(* Logix 5000 project; controller Motor_Test vendor 1 type 14 code 155 rev 32.11; software revision 32.01 *)

TASK MainTask (continuous, watchdog 500 ms) : MainProgram

MODULES
   Local : vendor 1 type 14 code 155 (PointIO 0, rev 32.11)
      Discrete_IO : Embedded (PointIO 1, rev 32.11, Output RPI 20 ms)
END_MODULES

VAR_GLOBAL   (* controller tags *)
   Empty : BOOL;
   Full : BOOL;
   Level : COUNTER := (PRE := 3, ACC := 1);
   LoadBegin : BOOL;
   LoadDone : BOOL;
   MoveSlots : DINT;
   OPC : BOOL;
   Slot : COUNTER := (PRE := 20, ACC := 1);
   TotalSteps : COUNTER := (PRE := 200);
END_VAR

PROGRAM MainProgram   (* main routine MainRoutine *)
VAR
   Begin_Step : BOOL;
   Change : BOOL;
   Count : COUNTER := (PRE := 10);
   DIR_Change : BOOL;
   Direction_CCW : ALIAS FOR Local:1:O.Data.1;
   During : BOOL;
   End_Step : BOOL;
   GoToStart : BOOL;
   High_Time : TIMER := (PRE := 50);
   High_Time_Temp : TIMER := (PRE := 500, ACC := 250);
   Increment : BOOL;
   LoadAccum : BOOL;
   LoadCount : INT;
   LoadCounter : COUNTER := (PRE := 1000);
   LoadHighTime : TIMER := (PRE := 50);
   Loading : BOOL;
   LoadLowTime : TIMER := (PRE := 50);
   LoadStepBegin : BOOL;
   LoadStepEnd : BOOL;
   Low_Time : TIMER := (PRE := 50);
   OPC_Test : BOOL;
   Pulse_Temp : BOOL;
   Step_Count : INT;
   Step_CW : ALIAS FOR Local:1:O.Data.0;
   Step_Max : INT := 10;
   Test_Done : BOOL;
   Test_Start : BOOL;
END_VAR

ROUTINE MainRoutine   (* ladder *)
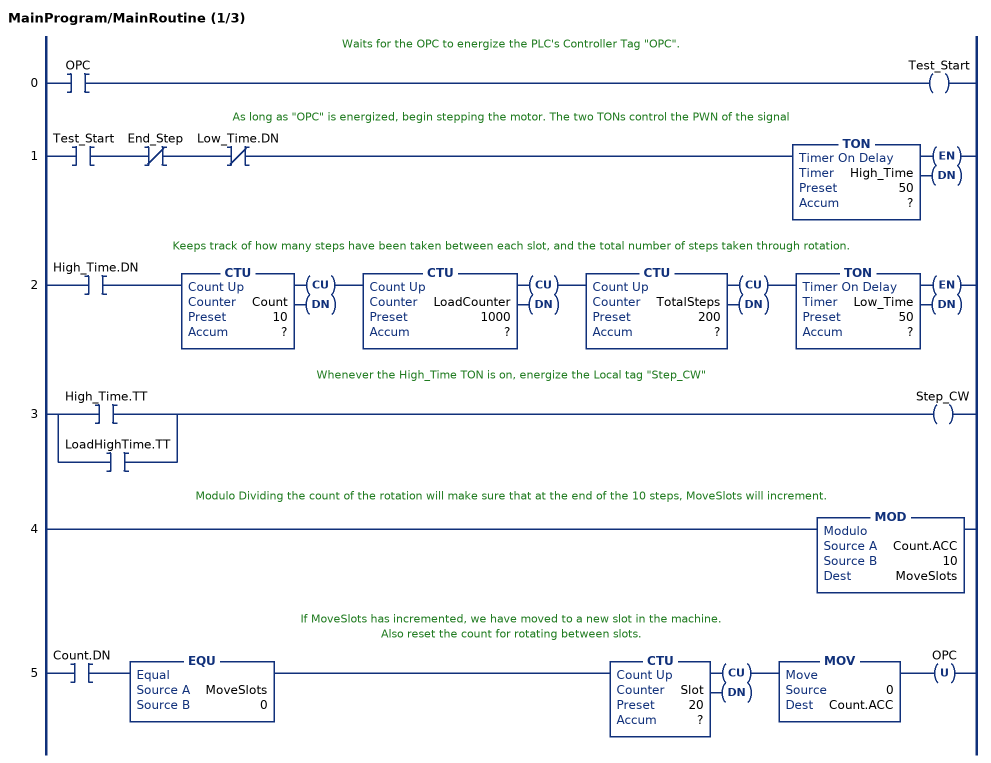
   // Waits for the OPC to energize the PLC's Controller Tag "OPC".
   0: XIC(OPC)OTE(Test_Start);
   // As long as "OPC" is energized, begin stepping the motor. The two TONs control the PWN of the signal
   1: XIC(Test_Start)XIO(End_Step)XIO(Low_Time.DN)TON(High_Time,?,?);
   // Keeps track of how many steps have been taken between each slot, and the total number of steps taken through rotation.
   2: XIC(High_Time.DN)CTU(Count,?,?)CTU(LoadCounter,?,?)CTU(TotalSteps,?,?)TON(Low_Time,?,?);
   // Whenever the High_Time TON is on, energize the Local tag "Step_CW"
   3: [XIC(High_Time.TT) ,XIC(LoadHighTime.TT) ]OTE(Step_CW);
   // Modulo Dividing the count of the rotation will make sure that at the end of the 10 steps, MoveSlots will increment.
   4: MOD(Count.ACC,10,MoveSlots);
   // If MoveSlots has incremented, we have moved to a new slot in the machine.
   // Also reset the count for rotating between slots.
   5: XIC(Count.DN)EQU(MoveSlots,0)CTU(Slot,?,?)MOV(0,Count.ACC)OTU(OPC);
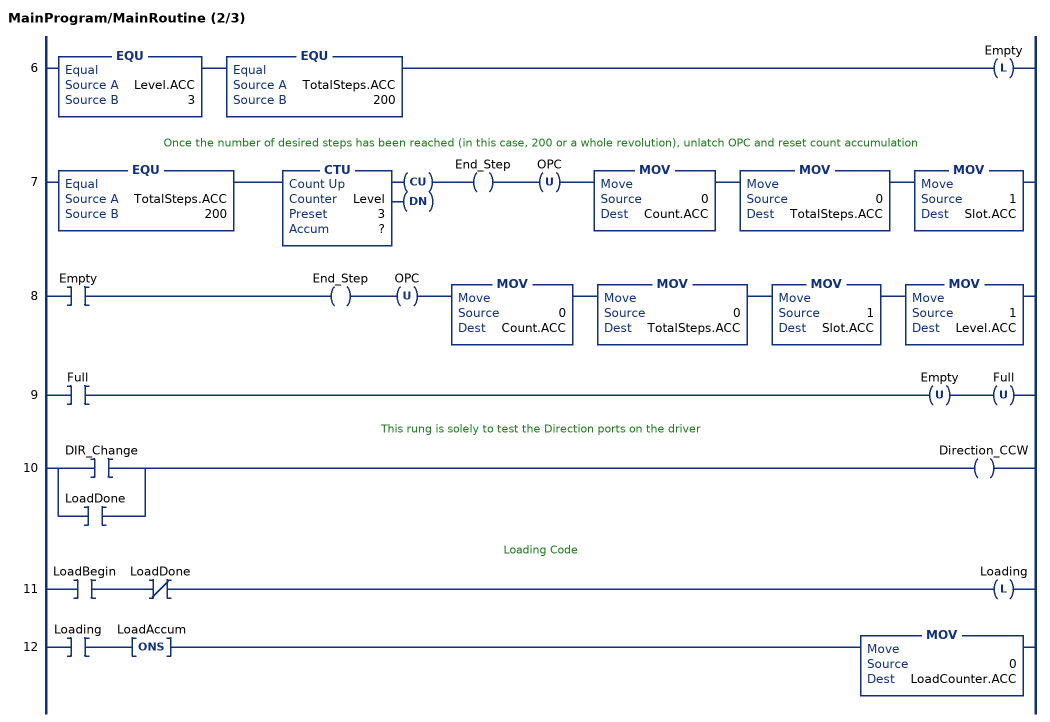
   6: EQU(Level.ACC,3)EQU(TotalSteps.ACC,200)OTL(Empty);
   // Once the number of desired steps has been reached (in this case, 200 or a whole revolution), unlatch OPC and reset count accumulation
   7: EQU(TotalSteps.ACC,200)CTU(Level,?,?)OTE(End_Step)OTU(OPC)MOV(0,Count.ACC)MOV(0,TotalSteps.ACC)MOV(1,Slot.ACC);
   8: XIC(Empty)OTE(End_Step)OTU(OPC)MOV(0,Count.ACC)MOV(0,TotalSteps.ACC)MOV(1,Slot.ACC)MOV(1,Level.ACC);
   9: XIC(Full)OTU(Empty)OTU(Full);
   // This rung is solely to test the Direction ports on the driver
   10: [XIC(DIR_Change) ,XIC(LoadDone) ]OTE(Direction_CCW);
   // Loading Code
   11: XIC(LoadBegin)XIO(LoadDone)OTL(Loading);
   12: XIC(Loading)ONS(LoadAccum)MOV(0,LoadCounter.ACC);
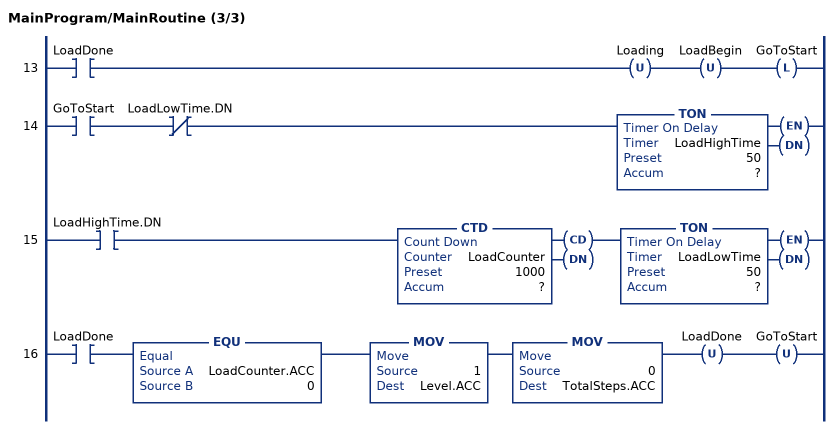
   13: XIC(LoadDone)OTU(Loading)OTU(LoadBegin)OTL(GoToStart);
   14: XIC(GoToStart)XIO(LoadLowTime.DN)TON(LoadHighTime,?,?);
   15: XIC(LoadHighTime.DN)CTD(LoadCounter,?,?)TON(LoadLowTime,?,?);
   16: XIC(LoadDone)EQU(LoadCounter.ACC,0)MOV(1,Level.ACC)MOV(0,TotalSteps.ACC)OTU(LoadDone)OTU(GoToStart);
END_ROUTINE
END_PROGRAM
